// TIA Portal V16 export
// export: Created 2024-09-05T17:39:16.0023034Z, ExportSetting WithDefaults, DisplayName Totally Integrated Automation Portal, DisplayVersion V16 Update 6, DisplayName TIA Portal Version Control Interface, DisplayVersion V16 Update 2, DisplayName TIA Portal Openness, DisplayVersion V16 Update 6, DisplayName STEP 7 Professional, DisplayVersion V16 Update 6, DisplayName STEP 7 Safety, DisplayVersion V16, DisplayName WinCC Advanced, DisplayVersion V16 Update 6
ORGANIZATION_BLOCK "OB_IO_AccessError"   // OB122, LAD, IOAccessError
{ S7_Optimized_Access := 'TRUE' }
VERSION : 0.1
// stored: IsIECCheckEnabled false, SetENOAutomatically false
   VAR_INPUT
      BlockNr : UInt;   // Number of causing block
      Reaction : USInt;   // 0:ignore, 1:substitute, 2:skip
      Fault_ID : Byte;   // 16#42:reading, 16#43:writing
      BlockType : USInt;   // 16#01:OB, 16#02:FC, 16#03:FB, 16#04:SFC, 16#05:SFB, 16#06:DB: Type of block causing the error
      Area : USInt;   // 16#81:I, 16#82:Q: IO area where the IOaccess error occured
      DBNr : DB_ANY;   // Reserved for system
      Csg_OBNr : OB_ANY;   // Number of OB causing the error
      Csg_Prio : USInt;   // Priority of OB causing the error
      Width : USInt;   // 0:bit, 1:byte, 2:word, 3:dword, 4:lword
   END_VAR
BEGIN
END_ORGANIZATION_BLOCK
